// TwinCAT 3 PLC project Untitled1
// ProgramVersion: 3.1.4023.0
// libraries:
//   Tc2_SerialCom, * (Beckhoff Automation GmbH)
//   Tc2_Standard, * (Beckhoff Automation GmbH)
//   Tc2_System, * (Beckhoff Automation GmbH)
//   Tc3_Module, * (Beckhoff Automation GmbH)
// project tree:
//   / PRG_10ms.TcPOU, Task_10ms.TcTTO
// real-time tasks:
//   TASK Task 10ms: cycle T#10ms, priority 3, ADS port 353

CONFIGURATION Untitled1
    RESOURCE PLC ON TwinCAT3
        TASK Task_10ms(INTERVAL := T#10ms, PRIORITY := 3);
        PROGRAM PRG_10ms WITH Task_10ms : PRG_10ms;
    END_RESOURCE
END_CONFIGURATION

// ---- PRG_10ms.TcPOU
PROGRAM PRG_10ms
VAR
	fbVirtualCOM							:SerialLineControlADS;
	fbComRec								:ReceiveData;
	fbComSend							:SendData;
	Delay									:TON;
	
	stCOMSerialConfig					:ComSerialConfig;	
	TXBuffer,RXBuffer					:ComBuffer;	
	aDataRec								:ARRAY[0..19] OF BYTE;
	aDataSend								:ARRAY[0..19] OF BYTE;
	bInit										:BOOL := TRUE;
END_VAR

stCOMSerialConfig.ComPort := 1;
stCOMSerialConfig.Baudrate := 9600;
stCOMSerialConfig.Parity := PARITY_EVEN;
stCOMSerialConfig.DataBits := 7;
stCOMSerialConfig.StopBits := STOPBITS_ONE;

fbVirtualCOM(
	Connect:= bInit, 
	SerialCfg:= stCOMSerialConfig, 
	NetId:= , 
	Timeout:= , 
	TxBuffer:= TXBuffer, 
	RxBuffer:= RXBuffer, 
	PortOpened=> , 
	Error=> , 
	ErrorID=> , 
	Busy=> , 
	TxBufCount=> , 
	RxBufCount=> );

Delay(IN:=NOT Delay.Q, PT := T#500MS);	
IF Delay.Q AND fbVirtualCOM.PortOpened THEN	
fbComSend(
	pSendData:= ADR(aDataSend), 
	Length:= SIZEOF(aDataSend), 
	Busy=> , 
	Error=> , 
	TXbuffer:= TXBuffer);	
END_IF
	
fbComRec(
	pPrefix:= , 
	LenPrefix:= , 
	pSuffix:= , 
	LenSuffix:= , 
	pReceiveData:= ADR(aDataRec), 
	SizeReceiveData:= SIZEOF(aDataRec), 
	Timeout:= , 
	Reset:= , 
	DataReceived=> , 
	busy=> , 
	Error=> , 
	RxTimeout=> , 
	LenReceiveData=> , 
	RXbuffer:= RXBuffer);

END_PROGRAM
